INTERFACE IExecution

METHOD Abort 
VAR_INPUT
END_VAR
END_METHOD

PROPERTY Aborted : BOOL
GET
END_GET
END_PROPERTY

PROPERTY Busy : BOOL
GET
END_GET
END_PROPERTY

PROPERTY Done : BOOL
GET
END_GET
END_PROPERTY

PROPERTY Error : BOOL
GET
END_GET
END_PROPERTY

PROPERTY ErrorId : UDINT
GET
END_GET
END_PROPERTY

PROPERTY Event_OnAbort : IEvent_ExecutionAborted
GET
END_GET
SET
END_SET
END_PROPERTY

PROPERTY Event_OnError : IEvent_ExecutionFailed
GET
END_GET
SET
END_SET
END_PROPERTY

PROPERTY Ready : BOOL
GET
END_GET
END_PROPERTY

METHOD Start : BOOL // returns TRUE if start request accepted (i.e State was Ready)
VAR_INPUT
END_VAR
END_METHOD

PROPERTY Starting : BOOL
GET
END_GET
END_PROPERTY

END_INTERFACE

(* stored: Version 1.1.0.1, ProductVersion 3.1.4024.3
   Itf IExecution: Id {2e2a9e90-2894-0caa-065e-86441183945f}
   Folder Methods: Id {4df2c49f-ecc5-41ac-a5f7-eb029ec847e7}
   Folder Properties: Id {1c6ea236-5ceb-43e5-bff2-34be35cf4670}
   Method Abort: Id {b913466c-26cf-0433-3b1e-51d91dedf168}
   Property Aborted: Id {b7d26468-ca45-08f2-25c2-2b915fb1a844}
   Get Get: Id {be2f86db-03f4-0428-2f88-5ded69f81209}
   Property Busy: Id {d4a7cc39-4b24-0b42-34b2-23d7b4599e03}
   Get Get: Id {ceae9d64-49ec-0008-0148-f7166e58a1e7}
   Property Done: Id {2bbbaca9-b4d7-0d31-1258-b75be134c5eb}
   Get Get: Id {4494e71e-066e-0cd0-0c21-ed633b55e85d}
   Property Error: Id {6f251179-ad69-092d-3e43-f4ea0910b03d}
   Get Get: Id {dc5ebf11-9e17-0791-1406-b9a9821d248b}
   Property ErrorId: Id {e70455b0-dc4b-0c34-1045-912ff9a82ed9}
   Get Get: Id {165412e3-1334-0344-3d7c-308dc7ad915f}
   Property Event_OnAbort: Id {108d3cac-fea7-0fc6-3765-09ada2624a9f}
   Get Get: Id {0c859122-0665-0a0d-110a-73813ca72a9d}
   Set Set: Id {21cb0494-ddab-0238-25b8-e2d16103bf2e}
   Property Event_OnError: Id {4872962c-0ee1-0488-2d70-f904ff29f89c}
   Get Get: Id {48d29ccb-44f7-04d1-063e-d9c1902067b6}
   Set Set: Id {d4675863-1ff1-0f55-16c1-3a861c19f824}
   Property Ready: Id {5ebd299f-9d69-02d6-0b8a-aced692b2330}
   Get Get: Id {3242ed87-607d-0dcb-1c3b-dd5e7eefd132}
   Method Start: Id {28e25cff-ad88-0708-05e8-5a4e484e10dc}
   Property Starting: Id {66894140-e1e7-08c1-0ae0-ca0143dc7e44}
   Get Get: Id {9dec5dd7-35fd-0abe-3ad0-ec4af579a1e2} *)
